TYPE ST_AuditControl :
STRUCT
	bReadDB							:BOOL;
	bReadDBSize						:BOOL;

	bFilter							:BOOL;
	bClear							:BOOL;
	sFilter_Key						:STRING;
	dtFilter_From					:DT;
	dtFilter_To						:DT;
	sFilter_User					:STRING;
	enFilter_Event					:EN_BatchEvents;
	iViewFilter						:BOOL;
	
	bExport							:BOOL;
	sExportName						:STRING;
	
	bDelete							:BOOL;
	bSend							:BOOL;
	
	iProdSelectedProcess			:INT;
	iCleanSelectedProcess			:INT;
	iBatchSelectedProcess			:INT;
	
	bScanRecipeParams				:BOOL;
	bScanPhases						:BOOL;
END_STRUCT
END_TYPE

(* stored: Version 1.1.0.1, ProductVersion 3.1.4024.12
   DUT ST_AuditControl: Id {9ca6db73-5e80-4bac-b8e8-aa9e584d0c01} *)
